FUNCTION_BLOCK UA_SkillMux (* Serialises OPC UA method calls onto command events and routes the accept/reject answer back to the calling method's RSP *)
  (* Standard: 61499-2 *)
  (* Version 2.0, 2026-09-27, Project contributors, Filling cell reference model *)
  PACKAGE fillingcell;
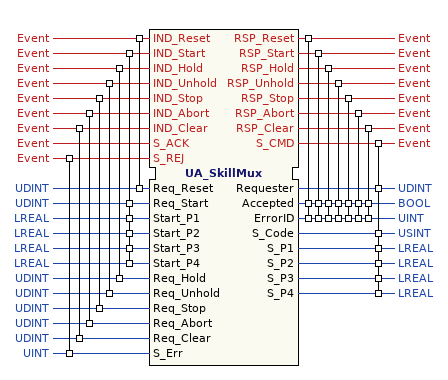
  EVENT_INPUT
    IND_Reset WITH Req_Reset;
    IND_Start WITH Req_Start, Start_P1, Start_P2, Start_P3, Start_P4;
    IND_Hold WITH Req_Hold;
    IND_Unhold WITH Req_Unhold;
    IND_Stop WITH Req_Stop;
    IND_Abort WITH Req_Abort;
    IND_Clear WITH Req_Clear;
    S_ACK;
    S_REJ WITH S_Err;
  END_EVENT
  EVENT_OUTPUT
    RSP_Reset WITH Accepted, ErrorID;
    RSP_Start WITH Accepted, ErrorID;
    RSP_Hold WITH Accepted, ErrorID;
    RSP_Unhold WITH Accepted, ErrorID;
    RSP_Stop WITH Accepted, ErrorID;
    RSP_Abort WITH Accepted, ErrorID;
    RSP_Clear WITH Accepted, ErrorID;
    S_CMD WITH Requester, S_Code, S_P1, S_P2, S_P3, S_P4;
  END_EVENT
  VAR_INPUT
    Req_Reset : UDINT;
    Req_Start : UDINT;
    Start_P1 : LREAL;
    Start_P2 : LREAL;
    Start_P3 : LREAL;
    Start_P4 : LREAL;
    Req_Hold : UDINT;
    Req_Unhold : UDINT;
    Req_Stop : UDINT;
    Req_Abort : UDINT;
    Req_Clear : UDINT;
    S_Err : UINT := 5;
  END_VAR
  VAR_OUTPUT
    Requester : UDINT;
    Accepted : BOOL;
    ErrorID : UINT;
    S_Code : USINT;
    S_P1 : LREAL;
    S_P2 : LREAL;
    S_P3 : LREAL;
    S_P4 : LREAL;
  END_VAR
  VAR
    Pending : USINT;
  END_VAR
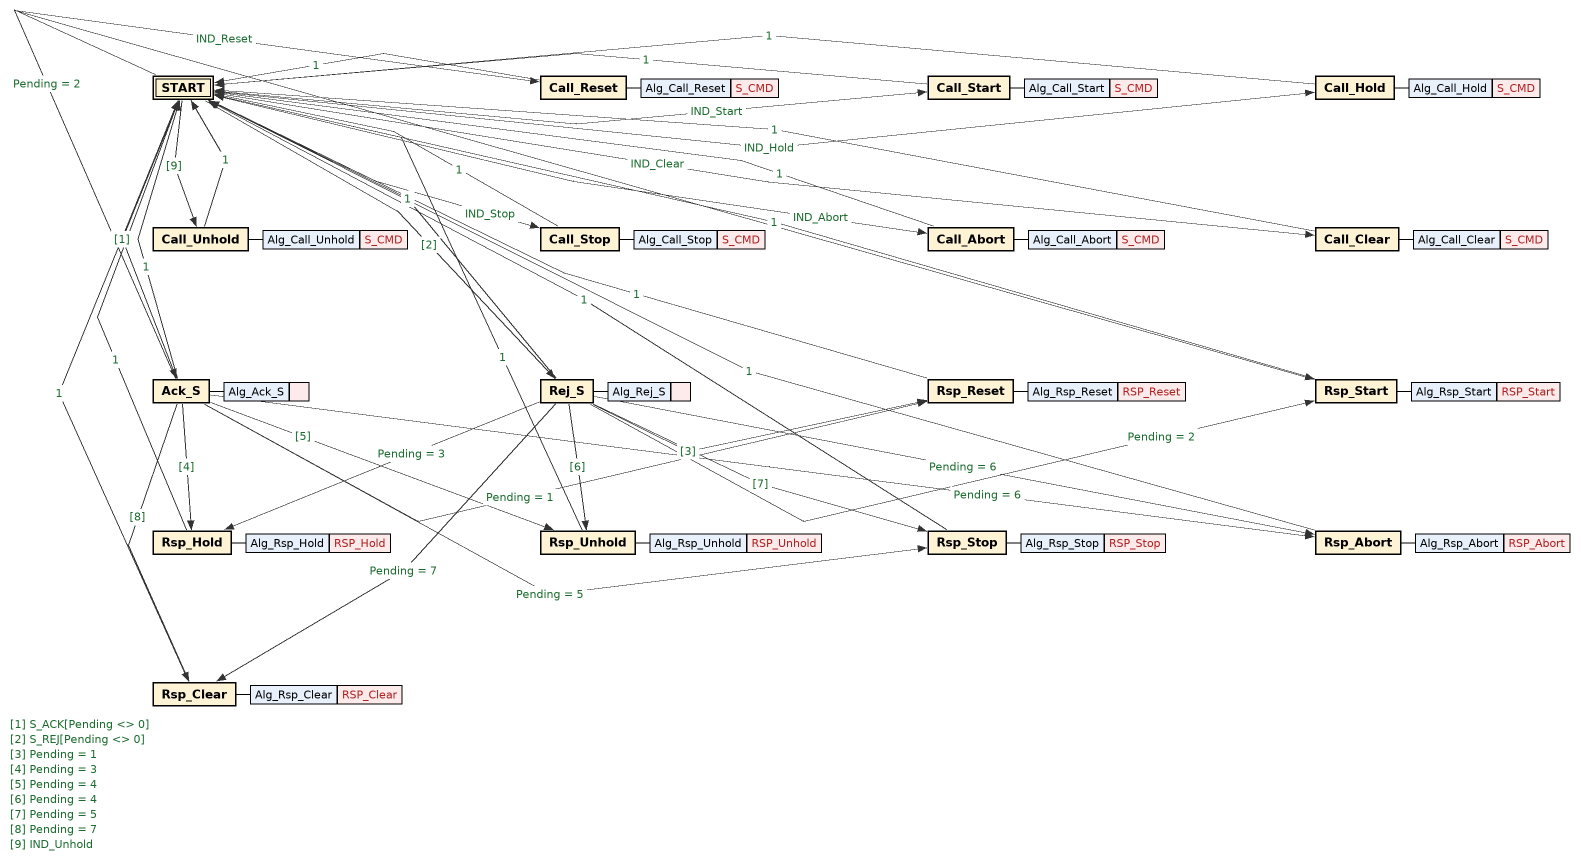
  EC_STATES
    START;
    Call_Reset : Alg_Call_Reset -> S_CMD;
    Call_Start : Alg_Call_Start -> S_CMD;
    Call_Hold : Alg_Call_Hold -> S_CMD;
    Call_Unhold : Alg_Call_Unhold -> S_CMD;
    Call_Stop : Alg_Call_Stop -> S_CMD;
    Call_Abort : Alg_Call_Abort -> S_CMD;
    Call_Clear : Alg_Call_Clear -> S_CMD;
    Ack_S : Alg_Ack_S;
    Rej_S : Alg_Rej_S;
    Rsp_Reset : Alg_Rsp_Reset -> RSP_Reset;
    Rsp_Start : Alg_Rsp_Start -> RSP_Start;
    Rsp_Hold : Alg_Rsp_Hold -> RSP_Hold;
    Rsp_Unhold : Alg_Rsp_Unhold -> RSP_Unhold;
    Rsp_Stop : Alg_Rsp_Stop -> RSP_Stop;
    Rsp_Abort : Alg_Rsp_Abort -> RSP_Abort;
    Rsp_Clear : Alg_Rsp_Clear -> RSP_Clear;
  END_STATES
  EC_TRANSITIONS
    START TO Call_Reset := IND_Reset;
    Call_Reset TO START := 1;
    START TO Call_Start := IND_Start;
    Call_Start TO START := 1;
    START TO Call_Hold := IND_Hold;
    Call_Hold TO START := 1;
    START TO Call_Unhold := IND_Unhold;
    Call_Unhold TO START := 1;
    START TO Call_Stop := IND_Stop;
    Call_Stop TO START := 1;
    START TO Call_Abort := IND_Abort;
    Call_Abort TO START := 1;
    START TO Call_Clear := IND_Clear;
    Call_Clear TO START := 1;
    START TO Ack_S := S_ACK[Pending <> 0];
    START TO Rej_S := S_REJ[Pending <> 0];
    Ack_S TO Rsp_Reset := Pending = 1;
    Rej_S TO Rsp_Reset := Pending = 1;
    Rsp_Reset TO START := 1;
    Ack_S TO Rsp_Start := Pending = 2;
    Rej_S TO Rsp_Start := Pending = 2;
    Rsp_Start TO START := 1;
    Ack_S TO Rsp_Hold := Pending = 3;
    Rej_S TO Rsp_Hold := Pending = 3;
    Rsp_Hold TO START := 1;
    Ack_S TO Rsp_Unhold := Pending = 4;
    Rej_S TO Rsp_Unhold := Pending = 4;
    Rsp_Unhold TO START := 1;
    Ack_S TO Rsp_Stop := Pending = 5;
    Rej_S TO Rsp_Stop := Pending = 5;
    Rsp_Stop TO START := 1;
    Ack_S TO Rsp_Abort := Pending = 6;
    Rej_S TO Rsp_Abort := Pending = 6;
    Rsp_Abort TO START := 1;
    Ack_S TO Rsp_Clear := Pending = 7;
    Rej_S TO Rsp_Clear := Pending = 7;
    Rsp_Clear TO START := 1;
    Ack_S TO START := 1;
    Rej_S TO START := 1;
  END_TRANSITIONS
  ALGORITHM Alg_Call_Reset IN ST:
Requester := Req_Reset;
S_Code := 1;
Pending := 1;
  END_ALGORITHM
  ALGORITHM Alg_Call_Start IN ST:
Requester := Req_Start;
S_Code := 2;
S_P1 := Start_P1;
S_P2 := Start_P2;
S_P3 := Start_P3;
S_P4 := Start_P4;
Pending := 2;
  END_ALGORITHM
  ALGORITHM Alg_Call_Hold IN ST:
Requester := Req_Hold;
S_Code := 3;
Pending := 3;
  END_ALGORITHM
  ALGORITHM Alg_Call_Unhold IN ST:
Requester := Req_Unhold;
S_Code := 4;
Pending := 4;
  END_ALGORITHM
  ALGORITHM Alg_Call_Stop IN ST:
Requester := Req_Stop;
S_Code := 5;
Pending := 5;
  END_ALGORITHM
  ALGORITHM Alg_Call_Abort IN ST:
Requester := Req_Abort;
S_Code := 6;
Pending := 6;
  END_ALGORITHM
  ALGORITHM Alg_Call_Clear IN ST:
Requester := Req_Clear;
S_Code := 7;
Pending := 7;
  END_ALGORITHM
  ALGORITHM Alg_Ack_S IN ST:
Accepted := TRUE;
ErrorID := 0;
  END_ALGORITHM
  ALGORITHM Alg_Rej_S IN ST:
Accepted := FALSE;
ErrorID := S_Err;
  END_ALGORITHM
  ALGORITHM Alg_Rsp_Reset IN ST:
Pending := 0;
  END_ALGORITHM
  ALGORITHM Alg_Rsp_Start IN ST:
Pending := 0;
  END_ALGORITHM
  ALGORITHM Alg_Rsp_Hold IN ST:
Pending := 0;
  END_ALGORITHM
  ALGORITHM Alg_Rsp_Unhold IN ST:
Pending := 0;
  END_ALGORITHM
  ALGORITHM Alg_Rsp_Stop IN ST:
Pending := 0;
  END_ALGORITHM
  ALGORITHM Alg_Rsp_Abort IN ST:
Pending := 0;
  END_ALGORITHM
  ALGORITHM Alg_Rsp_Clear IN ST:
Pending := 0;
  END_ALGORITHM
END_FUNCTION_BLOCK
